// TwinCAT 3 PLC project UnitTests
// ProgramVersion: 3.1.4022.7
// libraries:
//   lcls-twincat-motion, * (SLAC)
//   Tc2_Standard, * (Beckhoff Automation GmbH)
//   Tc2_System, * (Beckhoff Automation GmbH)
//   Tc3_Module, * (Beckhoff Automation GmbH)
//   TcUnit, * (www.tcunit.org)
// project tree:
//   GVLs/ SIM.TcGVL
//   / PlcTask.TcTTO
//   POUs/ MAIN.TcPOU
//   POUs/Motion/ FB_MotionRequest_Test.TcPOU
// (motion and I/O tree: see PLC project library)
// real-time tasks:
//   TASK PlcTask: cycle T#10ms, priority 20, ADS port 350
// variable links:

CONFIGURATION UnitTests
    RESOURCE PLC ON TwinCAT3
        TASK PlcTask(INTERVAL := T#10ms, PRIORITY := 20);
        PROGRAM MAIN WITH PlcTask : MAIN;
    END_RESOURCE
END_CONFIGURATION

// ---- GVLs/SIM.TcGVL
{attribute 'qualified_only'}
VAR_GLOBAL
    stBasicMotor: DUT_MotionStage;
END_VAR

// ---- POUs/MAIN.TcPOU
PROGRAM MAIN
VAR
    fbMotion: FB_MotionStage;
    fbMotionRequest_Test: FB_MotionRequest_Test;
END_VAR

fbMotion(stMotionStage:=SIM.stBasicMotor);
TcUnit.RUN();

END_PROGRAM

// ---- POUs/Motion/FB_MotionRequest_Test.TcPOU
FUNCTION_BLOCK FB_MotionRequest_Test EXTENDS TcUnit.FB_TestSuite
(*
    Verify that FB_MotionRequest works and is a suitable
    test proxy for FB_MotionStage
*)
VAR
    fbMotionSettings: FB_MotionStageSim_Settings;
    fbMotionReset: FB_MotionStage_Reset;
    fbMotionRequest: FB_MotionRequest;
    tonTimeout: TON;
    fGoal: LREAL := 50;
    nStep: INT := SETUP;
END_VAR
VAR CONSTANT
    SETUP: INT := 0;
    RUN: INT := 1;
    CHECK: INT := 2;
END_VAR

CASE nStep OF
    SETUP:
        TEST('FB_MotionRequest Basic Motion');
        fbMotionSettings(stMotionStage:=SIM.stBasicMotor);
        fbMotionReset(
            stMotionStage:=SIM.stBasicMotor,
            bExecute:=TRUE);
        IF fbMotionReset.bDone THEN
            AssertFalse(
                Condition:=SIM.stBasicMotor.bError,
                Message:='DUT_MotionStage had an error before we started!');
            fGoal := SIM.stBasicMotor.stAxisStatus.fActPosition + fGoal;
            nStep := RUN;
        END_IF
    RUN:
        fbMotionRequest(
            stMotionStage:=SIM.stBasicMotor,
            bExecute:=TRUE,
            fPos:=fGoal,
            fVel:=1000);

        tonTimeout(
            IN:=TRUE,
            PT:=T#1s);

        IF fbMotionRequest.bDone THEN
            nStep := CHECK;
        ELSIF tonTimeout.Q THEN
            AssertTrue(
                Condition:=FALSE,
                Message:='Timeout during basic motion test!');
            nStep := CHECK;
        END_IF
    CHECK:
        AssertEquals(
            Expected:=fGoal,
            Actual:=SIM.stBasicMotor.stAxisStatus.fActPosition,
            Message:='Failed to reach destination during basic motion test');
        AssertFalse(
            Condition:=fbMotionRequest.bError,
            Message:='FB_MotionRequest had an error during basic motion test');
        AssertFalse(
            Condition:=SIM.stBasicMotor.bError,
            Message:='DUT_MotionStage had an error during basic motion test');
        TEST_FINISHED();
END_CASE

END_FUNCTION_BLOCK
